Staubli VAL3: SetSpeed.pgx

program SetSpeed(num value)
begin
  //*******************************************************************************
  //*   ______
  //*  / _____) /|
  //* | |      / /
  //* | | /\  / /
  //* | | \ \/ /  _      Copyright (c) KEOLABS, 2016
  //* | |  \__/  | |        http://www.keolabs.com
  //* | |________| |
  //*  \__________/
  //*
  //********************************************************************************
  //*@file          : SetSpeed
  //*@author        : Yves Ragot
  //*@version       : $Id: SetSpeed.pgx 1644 2017-01-24 08:08:07Z yves $
  //*@brief         : Change speed parameter
  //*
  //*******************************************************************************/

  if ((value > 0) and (value <= 10000))

      // max translation speed
      mNomSpeed.tvel = value

      // max rotation speed
      mNomSpeed.vel = value / 10
      if (mNomSpeed.vel) > 100
          mNomSpeed.vel = 100
      endIf
  else
      GeneralStatus = 101
      LastErrorCode = 0
  endIf

end
